// TIA Portal V17 export
// export: Created 2024-01-30T08:49:14.4069566Z, ExportSetting WithDefaults, DisplayName Totally Integrated Automation Portal, DisplayVersion V17 Update 6, DisplayName TIA Portal Openness, DisplayVersion V17 Update 6, DisplayName TIA Portal Version Control Interface, DisplayVersion V17, DisplayName STEP 7 Professional, DisplayVersion V17 Update 6, DisplayName STEP 7 Safety, DisplayVersion V17 Update 6, DisplayName WinCC Advanced, DisplayVersion V17 Update 6
DATA_BLOCK "DB_ScanData"   // DB5
{ S7_Optimized_Access := 'TRUE' }
VERSION : 0.1
// stored: AutoNumber true, DBAccessibleFromOPCUA true, DBAccessibleFromWebserver true, IsOnlyStoredInLoadMemory false, IsRetainMemResEnabled false, IsWriteProtectedInAS false, MemoryReserve 100
   VAR
      ST01_MessGewichtMasse : Struct
         Request_for_Scan : Bool;
         DatenVorhanden : Bool;
         "Tray+Zelle" : Array[1..1, 1..1] of "UDT_ProGloveScanDat";
      END_STRUCT;
      ST02_EOLMessungImpdanz : Struct
         Request_for_Scan : Bool;
         DatenVoranden : Bool;
         "Tray+Zelle" : Array[1..2, 1..6] of "UDT_ProGloveScanDat";
      END_STRUCT;
      ST03_Dichtigkeitspruefung : Struct
         Request_for_Scan : Bool;
         DatenVoranden : Bool;
         "Tray+Zelle" : Array[1..1, 1..1] of "UDT_ProGloveScanDat";
      END_STRUCT;
      ST04_Degassing : Struct
         Request_for_Scan : Bool;
         DatenVorhanden : Bool;
         "Tray+Zelle" : Array[1..1, 1..1] of "UDT_ProGloveScanDat";
      END_STRUCT;
      ST05_Formierung : Struct
         Request_for_Scan : Bool;
         DatenVorhanden : Bool;
         Schrank : Array[1..2] of "UDT_Formierung";
      END_STRUCT;
      ST06_Soaking : Struct
         Request_for_Scan : Bool;
         DatenVorhanden : Bool;
         Schrank : Array[1..4] of "UDT_Formierung";
      END_STRUCT;
      ST07_Aging : Struct
         Request_for_Scan : Bool;
         DatenVorhanden : Bool;
         Schrank : Array[1..30] of "UDT_Aging";
      END_STRUCT;
      ST08_MobileOCVMessung : Struct
         Request_for_Scan : Bool;
         DatenVorhanden : Bool;
         "Tray+Zelle" : Array[1..1, 1..6] of "UDT_ProGloveScanDat";
      END_STRUCT;
   END_VAR
BEGIN
END_DATA_BLOCK
